PROGRAM INTERNAL PRG_Test
VAR
	fbContextBuilder_Test	: FB_ContextBuilder_Test;

	fbLog			: FB_Log;

	fbScope			: FB_ScopedContext;
	bLog			: BOOL;
	bArg1			: BOOL;
	nArg2			: INT;
	sArg3			: STRING;


END_VAR

TcUnit.RUN();

IF _TaskInfo[GETCURTASKINDEXEX()].FirstCycle THEN
	// For Remote TC-OTel Server change the AMS net ID and configure a route
	PRG_TaskLog.Init('10.10.10.10.1.1');
	F_Log(E_LogLevel.eInfo, 'SPS Task gestartet.').CreateLog();
END_IF

fbLog.LoggerContext.AddInt('logger', 42);

IF bLog THEN
	bLog := FALSE;
	F_Log(E_LogLevel.eDebug, 'Foobar').CreateLog();
	F_Log(E_LogLevel.eInfo, '{0}, {1}, {2}')
		.WithAnyArg(bArg1)
		.WithAnyArg(nArg2)
		.WithAnyArg(sArg3)
		.CreateLog();

	fbLog.Info('barbaz {bLog}')
		.WithAnyArg(bLog)
		.CreateLog();
END_IF

PRG_TaskLog.Call();

END_PROGRAM

(* stored: Version 1.1.0.1, ProductVersion 3.1.4026.18
   POU PRG_Test: Id {e5eebc94-2583-419e-a5ae-15055f39621e}, SpecialFunc None *)
